(*
Geographic Position
----------------

Overview
================

Represents a geodetic (or geocentric) position with latitude, longitude, and elevation (above the ellipsoid).
*)
FUNCTION_BLOCK GeoPosition
VAR_INPUT
END_VAR
VAR_OUTPUT
END_VAR
VAR
	Latitude_  : LREAL;//radians north of equator
	Longitude_ : LREAL;//radians east of meridian
	Elevation_ : LREAL;//m above ellipsoid
END_VAR

METHOD PUBLIC Clear
VAR_INPUT
END_VAR
Latitude_ := 0;
Longitude_ := 0;
Elevation_ := 0;
END_METHOD

METHOD PUBLIC CopyFrom
VAR_INPUT
	P : GeoPosition;
END_VAR
Latitude_ := P.LatitudeRad;
Longitude_ := P.LongitudeRad;
Elevation_ := P.Elevation;
END_METHOD

PROPERTY PUBLIC Elevation : LREAL
GET
Elevation := Elevation_;
END_GET
SET
Elevation_ := Elevation;
END_SET
END_PROPERTY

METHOD PUBLIC GetCartesianPosition : Vector3
VAR_INPUT
	Ref : REFERENCE TO GeoEllipsoid := GeoEllipsoids.WGS84;
END_VAR
IF NOT(__ISVALIDREF(Ref)) THEN
	GetCartesianPosition := GeoEllipsoids.WGS84.GetCartesianFromGeodetic(THIS^);
ELSE
	GetCartesianPosition := Ref.GetCartesianFromGeodetic(THIS^);
END_IF;
END_METHOD

//Gets the relative position of the supplied GeoPosition, considering this GeoPosition as an ENU tangent reference frame
METHOD PUBLIC GetRelativePosition : Vector3
VAR_INPUT
	P : GeoPosition;
	Ref : REFERENCE TO GeoEllipsoid := GeoEllipsoids.WGS84;
END_VAR
VAR
	EnuInEcef : HMatrix;
END_VAR
EnuInEcef := GetTangentEnuTransform(Ref);
GetRelativePosition := EnuInEcef.GetTransformedVector3Reverse(P.GetCartesianPosition(Ref));
END_METHOD

METHOD PUBLIC GetTangentEnuPose : GeoPose
VAR_INPUT
	Ref : REFERENCE TO GeoEllipsoid := GeoEllipsoids.WGS84;
END_VAR
GetTangentEnuPose.SetFromEcefTransformation(GetTangentEnuTransform(Ref),Ref);
END_METHOD

METHOD PUBLIC GetTangentEnuRotation : RMatrix
VAR_INPUT
	Ref : REFERENCE TO GeoEllipsoid := GeoEllipsoids.WGS84;
END_VAR
IF NOT(__ISVALIDREF(Ref)) THEN
	GetTangentEnuRotation := GeoEllipsoids.WGS84.GetTangentEnurotation(THIS^);
ELSE
	GetTangentEnuRotation := Ref.GetTangentEnurotation(THIS^);
END_IF
END_METHOD

METHOD PUBLIC GetTangentEnuTransform : HMatrix
VAR_INPUT
	Ref : REFERENCE TO GeoEllipsoid := GeoEllipsoids.WGS84;
END_VAR
IF NOT(__ISVALIDREF(Ref)) THEN
	GetTangentEnuTransform := GeoEllipsoids.WGS84.GetTangentEnuTransform(THIS^);
ELSE
	GetTangentEnuTransform := Ref.GetTangentEnuTransform(THIS^);
END_IF
END_METHOD

METHOD PUBLIC IsEqual : BOOL
VAR_INPUT
	P : REFERENCE TO GeoPosition;
END_VAR
IsEqual := IsNearlyEqual(P,0.0,0.0);
END_METHOD

METHOD PUBLIC IsNearlyEqual : BOOL
VAR_INPUT
	P : REFERENCE TO GeoPosition;
	PrecisionLatLon : LREAL;//radians
	PrecisionElevation : LREAL;//meters
END_VAR
IsNearlyEqual := ABS(P.LatitudeRad 		- LatitudeRad) 	<= PrecisionLatLon
             AND ABS(P.LongitudeRad 	- LongitudeRad) <= PrecisionLatLon
             AND ABS(P.Elevation 		- Elevation)	<= PrecisionElevation;
END_METHOD

PROPERTY PUBLIC LatitudeDeg : LREAL
GET
LatitudeDeg := 180.0 * Latitude_ /PI;
END_GET
SET
Latitude_ := PI * LatitudeDeg / 180.0;
END_SET
END_PROPERTY

PROPERTY PUBLIC LatitudeRad : LREAL
GET
LatitudeRad := Latitude_;
END_GET
SET
Latitude_ := LatitudeRad;
END_SET
END_PROPERTY

PROPERTY PUBLIC LongitudeDeg : LREAL
GET
LongitudeDeg := 180.0 * Longitude_ /PI;
END_GET
SET
Longitude_ := PI * LongitudeDeg / 180.0;
END_SET
END_PROPERTY

PROPERTY PUBLIC LongitudeRad : LREAL
GET
LongitudeRad := Longitude_;
END_GET
SET
Longitude_ := LongitudeRad;
END_SET
END_PROPERTY

METHOD PUBLIC SetFromCartesianPosition
VAR_INPUT
	V : Vector3;
	Ref : REFERENCE TO GeoEllipsoid;
END_VAR
VAR
	P : GeoPosition;
END_VAR
IF NOT(__ISVALIDREF(Ref)) THEN
	P := GeoEllipsoids.WGS84.GetGeodeticFromCartesian(V);
ELSE
	P := Ref.GetGeodeticFromCartesian(V);
END_IF
CopyFrom(P);
END_METHOD

METHOD PUBLIC SetFromComponentsDeg
VAR_INPUT
	Lat : LREAL;
	Lon : LREAL;
	El : LREAL;
END_VAR
LatitudeDeg := Lat;
LongitudeDeg := Lon;
Elevation := El;
END_METHOD

METHOD PUBLIC SetFromComponentsRad
VAR_INPUT
	Lat : LREAL;
	Lon : LREAL;
	El : LREAL;
END_VAR
LatitudeRad := Lat;
LongitudeRad := Lon;
Elevation := El;
END_METHOD

END_FUNCTION_BLOCK

(* stored: Version 1.1.0.1, ProductVersion 3.1.4024.9
   POU GeoPosition: Id {3af11355-6297-45a2-81e7-e3ba8de80095}, SpecialFunc None
   Folder Comparators: Id {a6df49ec-8996-434d-9ba6-f07e8fb8b6b7}
   Folder Helpers: Id {a898fd72-c3a8-4eaf-a197-d394a75c64fe}
   Folder Properties: Id {b7cf4284-fe56-4c36-a038-6435990ba7af}
   Folder Setters: Id {077d5114-78fa-4704-a6c3-9977056cbc5a}
   Method Clear: Id {2886a4c6-65cf-4e4a-8b87-9a8f58659c94}
   Method CopyFrom: Id {f42538b2-5d5a-42d4-9831-f395b8a59545}
   Property Elevation: Id {0a35baa3-1998-4c15-9742-43e0b8bbadf6}
   Get Get: Id {046cc5ea-a770-421a-bb1f-ad84db69148c}
   Set Set: Id {726bd732-8e27-4780-9d0c-f34f7df65e50}
   Method GetCartesianPosition: Id {c912fb69-b38e-4243-9dfa-151630fe823b}
   Method GetRelativePosition: Id {38805414-8032-4a19-a7fe-1523f39abb6b}
   Method GetTangentEnuPose: Id {fc67d3d8-12a4-46a3-8c72-f98a475d1072}
   Method GetTangentEnuRotation: Id {0af28ec9-5cf4-4531-856b-f760d4432ef7}
   Method GetTangentEnuTransform: Id {6c9c138d-3993-41c3-ad94-8f80f5c42f1b}
   Method IsEqual: Id {f18eb5d7-5a74-4649-8b7c-157f6655d827}
   Method IsNearlyEqual: Id {aa31bf7f-c28c-42b9-bc7f-9674c88e4763}
   Property LatitudeDeg: Id {ca76519e-ec08-4b92-86d5-8bcb86ec81ef}
   Get Get: Id {34bf9114-ffeb-42d1-9415-01337a15b981}
   Set Set: Id {3a8c8ca2-ee71-4ba5-9e46-f592f7f30627}
   Property LatitudeRad: Id {57917cbc-cae3-41ce-9a84-b7df5edb7322}
   Get Get: Id {ff87d137-9a83-4d69-93dc-8e2ad76693b0}
   Set Set: Id {7eca666d-736b-42b7-8bbc-aabcb2c49d4a}
   Property LongitudeDeg: Id {2bd865c8-e687-4487-b76e-c00ac3f628fc}
   Get Get: Id {9d388086-5deb-44a5-b974-2d9a55d286a9}
   Set Set: Id {5f0c9740-65c9-43c6-bbaf-f8b117ca798b}
   Property LongitudeRad: Id {b3ce4649-d336-472a-9c47-bffc37a3d5f5}
   Get Get: Id {30e343d8-81a8-447c-afee-33ee57b92e1c}
   Set Set: Id {65ac29d7-4868-4ca1-abba-72a48c6488f9}
   Method SetFromCartesianPosition: Id {048ddb8f-7491-418a-a8bf-7b2c0d60621f}
   Method SetFromComponentsDeg: Id {099b43f1-0625-4eba-84e3-19e82a3583b2}
   Method SetFromComponentsRad: Id {871b1570-e35a-48e7-acc1-bc64e9846475} *)
